// TIA Portal V18 export
// export: Created 2025-12-01T17:50:59.9784731Z, ExportSetting None, DisplayName Totally Integrated Automation Portal, DisplayVersion V18 Update 5, DisplayName TIA Portal Openness, DisplayVersion V18 Update 5, DisplayName TIA Portal Teamcenter Gateway, DisplayVersion V18, DisplayName TIA Portal Version Control Interface, DisplayVersion V18, DisplayName STEP 7 Professional, DisplayVersion V18 Update 5, DisplayName STEP 7 Safety, DisplayVersion V18, DisplayName WinCC Professional, DisplayVersion V18 Update 5
DATA_BLOCK "ST10_RecipeDB"   // DB1062
{ S7_Optimized_Access := 'FALSE' }
// stored: AutoNumber false
   VAR RETAIN
      Recipe : Struct   // System Defined=
         RecipeTag : String[50] := 'RecipeST10';   // 配方名称ID / System Defined=
         RecordName : String[50] := 'Product_1';   // 数据记录名称 / 配方名称ID
         PreConfigType : String[50] := 'Product_1';   // 待切换数据记录名称 / 数据记录名称
         Pulse : Bool := FALSE;   // 待切换数据记录名称
         Trigger : Bool := FALSE;   // 配方切换触发
         PosEdg : Bool := FALSE;   // 配方切换触发
         Alarm : Bool := FALSE;
         Ret : Bool := FALSE;
         Equal : Bool := TRUE;   // 换型OK标志位
         Pls : Bool := FALSE;   // 换型OK标志位
         "time" : Int := 0;
         Spare : Array[0..38] of Byte;
         DataRecord_TransferStatus : Int := 0;   // 数据记录传送状态
      END_STRUCT;
      ParameterElement : Struct
         TypeName : String[50] := 'Product_1';   // System Defined=
         TypeID : USInt := 1;   // System define= product type for parameters of servo ,press and so on
         FixtureID : Array[1..16] of Byte;
         A1_TableFixtureCode : Array[0..10] of String[128];   // 激光刻印程序号
         A2_TableFixtureCode : Array[0..10] of String[128];   // 贴标10号垂直气缸是否去工作位
         A1RingUnloadingFixtureCode : String[128] := 'SZ23055-OP010-E-Compresspr-ring1 cutting tool';
         E1LoadingNGFixtureCode : String[128] := 'SZ23055-OP010-E-Compressor-Left NG tooling-1';
         ShaftScanFixtureCode : String[128] := 'SZ23055-OP010-E-Compressor-shaft Rotating scanning tooling-1';
         B1PressFixtureCode : String[128] := 'SZ23055-OP010-E-Compressor-ring1 Below Positioning fixture -1';
         CGlueFixtureCode : String[128] := 'SZ23055-OP010-E-Compressor-Point adhesive tooling-1';
         B1PressCylFixtureCode : String[128] := 'SZ23055-OP010-E-Compressor-ring1 Upper pressing fixture-1';
         A2RingUnloadingFixtureCode : String[128] := 'SZ23055-OP010-E-Compresspr-ring2 cutting tool';
         E2UnloadingNGFixtureCode : String[128] := 'SZ23055-OP010-E-Compressor-Right NG tooling-1';
         B2PressFixtureCode : String[128] := 'SZ23055-OP010-E-Compressor-ring2 Below Positioning fixture -1';
         CGlueNGFixtureCode : String[128] := 'SZ23055-OP010-E-Compressor-NG middle shift tooling-1';
         B2PressCylFixtureCode : String[128] := 'SZ23055-OP010-E-Compressor-ring2 Upper pressing fixture-1';
         R1GripperFixtureCode : Array[0..6] of String[128];
         R2GripperFixtureCode : Array[0..6] of String[128];
         R3GripperFixtureCode : Array[0..6] of String[128];
         B1PressProgram : Int := 1;
         B2PressProgram : Int := 1;
         CGlueShaftIV3Program_1 : Word := 16#0001;
         CGlueShaftIV3Program_2 : Word := 16#0002;
         CGlueShaftIV3Program_3 : Word := 16#0003;
         CGlueShaftIV3Program_4 : Word := 16#0004;
         CGlueMagnetIV3Program : Word := 16#0001;
         CGlueProgram : Int := 1;
      END_STRUCT;
   END_VAR
BEGIN
   Recipe.Spare[0..38] := 16#00;
   ParameterElement.FixtureID[1] := 16#00;   // 工装编号
   ParameterElement.FixtureID[2..16] := 16#00;
   ParameterElement.A1_TableFixtureCode[0] := '';
   ParameterElement.A1_TableFixtureCode[1] := 'SZ23055-OP010-E-Compressor-ring1 Loading tooling-1';
   ParameterElement.A1_TableFixtureCode[2] := 'SZ23055-OP010-E-Compressor-ring1 Loading tooling-2';
   ParameterElement.A1_TableFixtureCode[3] := 'SZ23055-OP010-E-Compressor-ring1 Loading tooling-3';
   ParameterElement.A1_TableFixtureCode[4] := 'SZ23055-OP010-E-Compressor-ring1 Loading tooling-4';
   ParameterElement.A1_TableFixtureCode[5] := 'SZ23055-OP010-E-Compressor-ring1 Loading tooling-5';
   ParameterElement.A1_TableFixtureCode[6] := 'SZ23055-OP010-E-Compressor-ring1 Loading tooling-6';
   ParameterElement.A1_TableFixtureCode[7] := 'SZ23055-OP010-E-Compressor-ring1 Loading tooling-7';
   ParameterElement.A1_TableFixtureCode[8] := 'SZ23055-OP010-E-Compressor-ring1 Loading tooling-8';
   ParameterElement.A1_TableFixtureCode[9..10] := '';
   ParameterElement.A2_TableFixtureCode[0] := '';
   ParameterElement.A2_TableFixtureCode[1] := 'SZ23055-OP010-E-Compressor-ring2 Loading tooling-1';
   ParameterElement.A2_TableFixtureCode[2] := 'SZ23055-OP010-E-Compressor-ring2 Loading tooling-2';
   ParameterElement.A2_TableFixtureCode[3] := 'SZ23055-OP010-E-Compressor-ring2 Loading tooling-3';
   ParameterElement.A2_TableFixtureCode[4] := 'SZ23055-OP010-E-Compressor-ring2 Loading tooling-4';
   ParameterElement.A2_TableFixtureCode[5] := 'SZ23055-OP010-E-Compressor-ring2 Loading tooling-5';
   ParameterElement.A2_TableFixtureCode[6] := 'SZ23055-OP010-E-Compressor-ring2 Loading tooling-6';
   ParameterElement.A2_TableFixtureCode[7] := 'SZ23055-OP010-E-Compressor-ring2 Loading tooling-7';
   ParameterElement.A2_TableFixtureCode[8] := 'SZ23055-OP010-E-Compressor-ring2 Loading tooling-8';
   ParameterElement.A2_TableFixtureCode[9..10] := '';
   ParameterElement.R1GripperFixtureCode[0] := '';
   ParameterElement.R1GripperFixtureCode[1] := 'SZ23055-OP010-E-Compressor-robot1 ring1 Left clamping jaw tooling-1';
   ParameterElement.R1GripperFixtureCode[2] := 'SZ23055-OP010-E-Compressor-robot1 ring1 Right clamping jaw tooling-2';
   ParameterElement.R1GripperFixtureCode[3] := 'SZ23055-OP010-E-Compressor-robot1 shaft Left clamping jaw tooling-1';
   ParameterElement.R1GripperFixtureCode[4] := 'SZ23055-OP010-E-Compressor-robot1 shaft Right clamping jaw tooling-2';
   ParameterElement.R1GripperFixtureCode[5..6] := '';
   ParameterElement.R2GripperFixtureCode[0] := '';
   ParameterElement.R2GripperFixtureCode[1] := 'SZ23055-OP010-E-Compressor-robot2 shaft Right clamping jaw tooling-2';
   ParameterElement.R2GripperFixtureCode[2] := 'SZ23055-OP010-E-Compressor-robot2 shaft Left clamping jaw tooling-1';
   ParameterElement.R2GripperFixtureCode[3] := 'SZ23055-OP010-E-Compressor-robot2 magnet Left clamping jaw tooling-1';
   ParameterElement.R2GripperFixtureCode[4] := 'SZ23055-OP010-E-Compressor-robot2 magnet Right clamping jaw tooling-2';
   ParameterElement.R2GripperFixtureCode[5..6] := '';
   ParameterElement.R3GripperFixtureCode[0] := '';
   ParameterElement.R3GripperFixtureCode[1] := 'SZ23055-OP010-E-Compressor-robot3 ring2 Right clamping jaw tooling-2';
   ParameterElement.R3GripperFixtureCode[2] := 'SZ23055-OP010-E-Compressor-robot3 ring2 Left clamping jaw tooling-1';
   ParameterElement.R3GripperFixtureCode[3] := 'SZ23055-OP010-E-Compressor-robot3 shaft Left clamping jaw tooling-1';
   ParameterElement.R3GripperFixtureCode[4] := 'SZ23055-OP010-E-Compressor-robot3 shaft Right clamping jaw tooling-2';
   ParameterElement.R3GripperFixtureCode[5..6] := '';
END_DATA_BLOCK
